INTERFACE I_Command

METHOD execute
END_METHOD

END_INTERFACE

(* stored: Version 1.1.0.1
   Itf I_Command: Id {22b5179b-eb51-4fd7-b4b6-82d899b3d3ea}
   Method execute: Id {8bca204d-3e97-4e77-896e-d1bef3ecb3af} *)
